(* IEC 61131-3 sources: Generador-Horizontal-de-Oleaje/software/controller, 1 file *)

(* ---- wavewall-plc-code.st ---- *)
PROGRAM WaveWallController
VAR
    // Entradas analogicas
    aiWaveHeight      : REAL;   // Altura de ola (m)
    aiWavePeriod      : REAL;   // Periodo de ola (s)
    aiHydraulicPressure : REAL; // Presion hidraulica (bar)
    aiHydraulicFlow   : REAL;   // Caudal hidraulico (L/min)
    aiGeneratorRPM    : REAL;   // RPM generador
    aiGeneratorTemp   : REAL;   // Temperatura generador (C)

    // Entradas digitales
    diEmergencyStop   : BOOL;   // Parada de emergencia
    diGridConnected   : BOOL;   // Estado conexion a red

    // Salidas analogicas
    aoPumpDisplacement : REAL;  // Desplazamiento bomba (%)
    aoValvePosition   : REAL;   // Posicion valvula proporcional (%)

    // Salidas digitales
    doMainContactor   : BOOL;   // Contactor principal
    doGridSync        : BOOL;   // Sincronizacion con red
    doWarningLight    : BOOL;   // Luz de advertencia

    // Variables internas
    rPowerOutput      : REAL;   // Potencia instantanea (kW)
    rEnergyToday      : REAL;   // Energia diaria (kWh)
    iCycleCount       : INT;    // Contador de ciclos
    bMPPTEnable       : BOOL;   // Habilita MPPT
    rSetpointTorque   : REAL;   // Setpoint de torque (Nm)

    // Algoritmo predictivo
    arrWaveHistory    : ARRAY[1..60] OF REAL;
    iHistoryIndex     : INT;
    rPredictedPower   : REAL;
END_VAR

// Inicializacion
IF NOT bMPPTEnable THEN
    bMPPTEnable := TRUE;
    iCycleCount := 0;
    rEnergyToday := 0.0;
    FOR i := 1 TO 60 DO
        arrWaveHistory[i] := 0.0;
    END_FOR
END_IF

// Muestreo cada 100 ms
iCycleCount := iCycleCount + 1;

// Algoritmo MPPT adaptativo basado en periodo de ola
CASE TRUE OF
    aiWavePeriod < 5.0:
        aoPumpDisplacement := 65.0;  // Olas cortas, menor desplazamiento
    aiWavePeriod < 8.0:
        aoPumpDisplacement := 85.0;  // Olas medias, optimo
    ELSE:
        aoPumpDisplacement := 95.0;  // Olas largas, maxima captura
END_CASE

// Control de presion hidraulica
IF aiHydraulicPressure > 210.0 THEN
    aoValvePosition := aoValvePosition - 2.0;  // Derivar flujo
ELSIF aiHydraulicPressure < 180.0 THEN
    aoValvePosition := aoValvePosition + 2.0;  // Aumentar carga
END_IF
aoValvePosition := LIMIT(0.0, aoValvePosition, 100.0);

// Calculo de potencia
rPowerOutput := (aiHydraulicPressure * aiHydraulicFlow) / 600.0; // kW
rEnergyToday := rEnergyToday + (rPowerOutput * 0.1 / 3600.0); // kWh

// Algoritmo predictivo (ventana deslizante de 6 segundos)
arrWaveHistory[iHistoryIndex] := aiWaveHeight;
iHistoryIndex := iHistoryIndex + 1;
IF iHistoryIndex > 60 THEN iHistoryIndex := 1; END_IF

// Prediccion de potencia para los proximos 2 segundos
rPredictedPower := 0.0;
FOR i := 1 TO 20 DO
    rPredictedPower := rPredictedPower + arrWaveHistory[(iHistoryIndex - i + 60) MOD 60 + 1];
END_FOR
rPredictedPower := rPredictedPower / 20.0 * 12.0; // Factor de conversion empirico

// Logica de sincronizacion con red
IF diGridConnected AND NOT doGridSync THEN
    IF ABS(aiGeneratorRPM - 1500) < 10 THEN
        doGridSync := TRUE;
        doMainContactor := TRUE;
    END_IF
END_IF

// Protecciones
IF aiGeneratorTemp > 85.0 OR diEmergencyStop THEN
    doMainContactor := FALSE;
    doGridSync := FALSE;
    aoPumpDisplacement := 0.0;
    doWarningLight := TRUE;
ELSE
    doWarningLight := FALSE;
END_IF

// Comunicacion con Wave-Cloud (via Modbus TCP)
// Los datos se exponen en registros para ser leidos por el gateway
